// TIA Portal V18 export
// export: Created 2026-03-12T16:04:34.6094034Z, ExportSetting WithDefaults, DisplayName Totally Integrated Automation Portal, DisplayVersion V18 Update 5, DisplayName TIA Portal Openness, DisplayVersion V18 Update 5, DisplayName TIA Portal Version Control Interface, DisplayVersion V18, DisplayName SINAMICS Startdrive Advanced, DisplayVersion V18, DisplayName SINAMICS Startdrive G130, G150, S120, S150, SINAMICS MV, S210, DisplayVersion V18, DisplayName SINAMICS Startdrive G110M, G120, G120C, G120D, G120P, G115D, DisplayVersion V18, DisplayName STEP 7 Professional, DisplayVersion V18 Update 5, DisplayName STEP 7 Safety, DisplayVersion V18, DisplayName WinCC Professional, DisplayVersion V18 Update 5
FUNCTION_BLOCK "FB SUCÇÃO OK"   // FB15, LAD
TITLE = Function Block FB SUCÇÃO OK
{ S7_Optimized_Access := 'TRUE' }
VERSION : 0.1
// stored: AutoNumber true, IsIECCheckEnabled false, IsRetainMemResEnabled false, MemoryReserve 100, SetENOAutomatically false, UDAEnableTagReadback false
   VAR_INPUT
      REFERENCIA : Real;   // Referência analógica em relação à sucção da bomba
      CADASTRO_SUCÇAO_INSUFICIENTE : Real;   // Cadastro de nível/pressão insuficiente
      CADASTRO_TEMPO_RESET : Time;   // Cadastro do tempo para resetar o alarme de Pressão Insuficiente
   END_VAR
   VAR_OUTPUT
      SUCÇÃO_OK : Bool;   // Sucção OK para operação
   END_VAR
   VAR
      SUCCAO_INSUFICIENTE : Bool;   // Sucção Insuficiente para operação
      RESET_ALARME : IEC_TIMER;   // Reset alarme de Sucção Insuficiente
   END_VAR
BEGIN

REGION Network 1: Set e Reset da Referência de Sucção insuficiente
   // Se nível for menor que a referência do Reservatório SUCÇÃO INSUFICIENTE,  bomba não pode ligar.
   // Caso o Nivel seja maior que a refêrencia então, após tempo cadastrado a bomba está habita para ligar
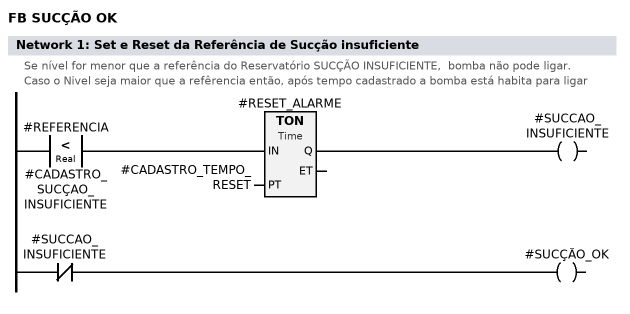
   RUNG wire#powerrail
      { S7_Templates := "SrcType := Real" } LT_Contact(in1 := #REFERENCIA, in2 := #CADASTRO_SUCÇAO_INSUFICIENTE)
      { S7_Templates := "time_type := Time" } #RESET_ALARME.TON(pt := #CADASTRO_TEMPO_RESET, et =>)
      Coil( #SUCCAO_INSUFICIENTE )
   END_RUNG
   RUNG wire#powerrail
      I_Contact( #SUCCAO_INSUFICIENTE )
      Coil( #SUCÇÃO_OK )
   END_RUNG
   // the same network as SCL:
   #RESET_ALARME.TON(IN := #REFERENCIA < #CADASTRO_SUCÇAO_INSUFICIENTE, PT := #CADASTRO_TEMPO_RESET);
   #SUCCAO_INSUFICIENTE := #RESET_ALARME.Q;
   #SUCÇÃO_OK := NOT #SUCCAO_INSUFICIENTE;
END_REGION
END_FUNCTION_BLOCK
